# EPICS autosave request: ip/ipApp/Db/PACE5000_settings.req
$(P)$(R)Units
$(P)$(R)Setpoint
$(P)$(R)TweakVal
$(P)$(R)SlewMode
$(P)$(R)Slew
$(P)$(R)ReadSettingsScan.SCAN
